TYPE ST_Tuning :
STRUCT
    nInfoData1 AT %I*: INT; // Mapped to EL7047 PDO InfoData 1 (e.g. Load)
    nInfoData2 AT %I*: INT; // Mapped to EL7047 PDO InfoData 2 (e.g. Power)
    bStall AT %I*: BOOL; // Mapped to EL7047 0x6010:08 (Stall)
END_STRUCT
END_TYPE

(* stored: Version 1.1.0.1
   DUT ST_Tuning: Id {42decf5b-5866-4f05-acc2-24ed83b2f4e4} *)
